FUNCTION_BLOCK FB_DiameterMovement EXTENDS FB_ObjectBase_V2
VAR_INPUT
//    Execute    :BOOL;   // True : This prog will start.
//    Abort      :BOOL;   // True : This prog will be abort.
//    Reset      :BOOL;   // True : This prog will be reset.
//    ObjectName :STRING; // Set this fb name(About it's action)
	
	bContinue:BOOL;
	
//	DiameterHorizontalCylinder 	:REFERENCE TO FB_Cylinder;	//測徑橫移氣壓缸
//	DiameterUpDownCylinder		:REFERENCE TO FB_Cylinder;	//測徑上下氣壓缸
//	DiameterClampCylinder		:REFERENCE TO FB_Cylinder; //測徑夾爪氣壓缸

	Cylinder : REFERENCE TO UNI_CylinderList;
	
END_VAR

VAR_OUTPUT
//    Busy    :BOOL;        // True : This prog is running.
//    Done    :BOOL;        // True : Command has been executed.
//    Aborted :BOOL;        // True : This prog is aborted.
//    Error   :BOOL;        // True : This prog has an error.
//    ErrorID :UINT;       // Output ErrorID
//    Status  :T_MaxString; // Output this prog status by string(255bytes)
	PickDone	:BOOL;
END_VAR

VAR
//    eState :E_MethodStatus_Basic;
//	uiExecutingStep : UDINT; // This var is used to been controll STATE_EXECUTING process.
//	uiResettingStep : UDINT;
//	uiAbortingStep : UDINT;
//	_Executed :BOOL; // Executing process completed.
//	_Error : BOOL; // FB has an error.
//	_ResetCompleted : BOOL; // FB resetting completed.
//	_AbortCompleted : BOOL; // FB aborting completed.
//	_Abort		: BOOL;
	strStatus	: STRING;
	uiResumeStep : UINT;
	tonDiameterTimeoutTwo :TON;
	
END_VAR

A00_BasicUnits();
SUPER^.A10_StateControl();

ACTION A00_BasicUnits:
tonDiameterTimeoutTwo(PT:=T#2S);
END_ACTION

METHOD GetModelState
VAR_OUTPUT
    xDone    :BOOL;
    xBusy    :BOOL;
    xError   :BOOL;
    xAborted :BOOL;
    iErrorID :UDINT;
	UniqueErrorCode : STRING;
END_VAR
xDone    := Done;
xBusy    := Busy;
xError   := Error;
xAborted := Abort;
iErrorID := ErrorID;
END_METHOD

METHOD GetName : STRING
GetName := ObjectName;
END_METHOD

METHOD  M_STATE_ABORTED
VAR_INPUT
END_VAR
ERROR :=TRUE;
Status := strStatus;

IF NOT Execute THEN
	eSTATE:=STATE_RESETTING;
END_IF

IF Execute AND Reset THEN
	uiExecutingStep :=uiResumeStep;
	eSTATE:=STATE_EXECUTING;
END_IF
END_METHOD

METHOD  M_STATE_ABORTING
VAR_INPUT
END_VAR
CASE uiAbortingStep OF
	
	
	9999:	_AbortCompleted:=TRUE;
END_CASE

IF _AbortCompleted THEN	
	eSTATE :=STATE_ABORTED;
END_IF
END_METHOD

METHOD  M_STATE_DONE
VAR_INPUT
END_VAR
Busy := FALSE;
Done:=TRUE;

IF NOT Execute THEN
	eSTATE:=STATE_RESETTING;
END_IF
END_METHOD

METHOD  M_STATE_DORMANT
VAR_INPUT
END_VAR
_Executed:=FALSE;
_Error	:=FALSE;
_Abort :=FALSE;
strStatus :='No Error';
uiResettingStep:=0;
uiExecutingStep :=0;
tonDiameterTimeoutTwo.IN:=FALSE;
Error := Busy := Done := FALSE;

IF Execute THEN
	eSTATE:=STATE_EXECUTING;
END_IF
END_METHOD

METHOD  M_STATE_ERROR
VAR_INPUT
END_VAR
ERROR :=TRUE;
Busy :=FALSE;
Done := FALSE;
Status := strStatus;
IF NOT Execute THEN	
eSTATE:=STATE_RESETTING;
END_IF
END_METHOD

METHOD  M_STATE_EXECUTING
VAR_INPUT
END_VAR
Busy :=TRUE;

CASE uiExecutingStep OF
	

0: //Standby todo : check 
	
		uiExecutingStep:=10;
10:
		
		IF Cylinder.List.fbUpCV_DiameterHoriz.xError THEN
			Cylinder.List.fbUpCV_DiameterHoriz.M_Reset();
		END_IF
		IF Cylinder.List.fbUpCV_DiameterVert.xError THEN
			Cylinder.List.fbUpCV_DiameterVert.M_Reset();
		END_IF
		IF Cylinder.List.fbUpCV_DiameterClamp.xError THEN
			Cylinder.List.fbUpCV_DiameterClamp.M_Reset();
		END_IF
		uiExecutingStep:=20;
		
20:
	Cylinder.List.fbUpCV_DiameterVert.M_Retract();
	IF Cylinder.List.fbUpCV_DiameterClamp.InFrontPosition THEN
		uiExecutingStep:=30;
	ELSE
		uiExecutingStep:=60;	
	END_IF
30:
	
	IF Cylinder.List.fbUpCV_DiameterVert.InRearPosition THEN
		Cylinder.List.fbUpCV_DiameterHoriz.M_Extend();
		uiExecutingStep:=40;
	END_IF
40:		
	IF Cylinder.List.fbUpCV_DiameterHoriz.InFrontPosition THEN
		Cylinder.List.fbUpCV_DiameterClamp.M_Retract();
		uiExecutingStep:=50;
	END_IF
50:	
	IF Cylinder.List.fbUpCV_DiameterClamp.InRearPosition THEN
		uiExecutingStep:=60;
	END_IF
	
60 : 
	Cylinder.List.fbUpCV_DiameterHoriz.M_Retract();
		uiExecutingStep:=70;
70:
	IF Cylinder.List.fbUpCV_DiameterHoriz.InRearPosition THEN
		uiExecutingStep:=1000;	
	END_IF
			
	

1000:// Pick to diameter camera position start: Clamp down
	Cylinder.List.fbUpCV_DiameterVert.M_Extend();
	uiExecutingStep:=1100;
	
1100:// wait clamp down
	tonDiameterTimeoutTwo.IN:=TRUE;
	IF 	Cylinder.List.fbUpCV_DiameterVert.InFrontPosition THEN
		tonDiameterTimeoutTwo.IN:=FALSE;
		uiExecutingStep:=1200;
	END_IF
	IF tonDiameterTimeoutTwo.Q THEN
		_Error :=TRUE;
		strStatus:='Cylinder.List.fbUpCV_DiameterVert MoveForward Timeout';
	END_IF
	
1200: // Clamp close
	Cylinder.List.fbUpCV_DiameterClamp.M_Extend();
	uiExecutingStep:=1300;

1300://wait clamp close
	tonDiameterTimeoutTwo.IN:=TRUE;
	IF 	Cylinder.List.fbUpCV_DiameterClamp.InFrontPosition THEN
		tonDiameterTimeoutTwo.IN :=FALSE;
		uiExecutingStep:=1400;
	END_IF
	IF tonDiameterTimeoutTwo.Q THEN
		_Error :=TRUE;
		strStatus:='Cylinder.List.fbUpCV_DiameterClamp M_Extend Timeout';
	END_IF
1400 : //Clamp up
	Cylinder.List.fbUpCV_DiameterVert.M_Retract();
	uiExecutingStep:=1500;	

1500:// wait clamp up
		tonDiameterTimeoutTwo.IN :=TRUE;
	IF 	Cylinder.List.fbUpCV_DiameterVert.InRearPosition THEN
		tonDiameterTimeoutTwo.IN :=FALSE;
		uiExecutingStep:=1600;
	END_IF
	IF tonDiameterTimeoutTwo.Q THEN
		_Error :=TRUE;
		strStatus:='Cylinder.List.fbUpCV_DiameterVert M_Retract Timeout';
	END_IF
1600: //Move horizontal
	Cylinder.List.fbUpCV_DiameterHoriz.M_Extend();
	uiExecutingStep:=1700;

1700://wait move horizontal
		tonDiameterTimeoutTwo.IN:=TRUE;
	IF 	Cylinder.List.fbUpCV_DiameterHoriz.InFrontPosition THEN
		tonDiameterTimeoutTwo.IN :=FALSE;
		uiExecutingStep:=1800;
	END_IF
		IF tonDiameterTimeoutTwo.Q THEN
		_Error :=TRUE;
		strStatus:='Cylinder.List.fbUpCV_DiameterHoriz M_Extend Timeout';
	END_IF

1800://Move down to diameter camera position
	Cylinder.List.fbUpCV_DiameterVert.M_Extend();
	uiExecutingStep:=1900;
	
1900:
		tonDiameterTimeoutTwo.IN:=TRUE;
	IF 	Cylinder.List.fbUpCV_DiameterVert.InFrontPosition THEN
		tonDiameterTimeoutTwo.IN :=FALSE;
		uiExecutingStep:=2000;
	END_IF	
	IF tonDiameterTimeoutTwo.Q THEN
		_Error :=TRUE;
		strStatus:='Cylinder.List.fbUpCV_DiameterVert M_Extend Timeout';
	END_IF

2000: 
	PickDone :=TRUE;
	IF bContinue THEN
		PickDone :=FALSE;
		uiExecutingStep:=5000;
	END_IF

5000: // Place needle back to box start
	Cylinder.List.fbUpCV_DiameterVert.M_Retract();
	uiExecutingStep:=5100;
	
5100:// wait clamp down
	tonDiameterTimeoutTwo.IN :=TRUE;
	IF 	Cylinder.List.fbUpCV_DiameterVert.InRearPosition THEN
		tonDiameterTimeoutTwo.IN :=FALSE;
		uiExecutingStep:=5200;
	END_IF
	IF tonDiameterTimeoutTwo.Q THEN
		_Error :=TRUE;
		strStatus:='Cylinder.List.fbUpCV_DiameterVert M_Retract Timeout';
	END_IF
	
5200: 
		Cylinder.List.fbUpCV_DiameterHoriz.M_Retract();
		uiExecutingStep := 5300;

5300:
		tonDiameterTimeoutTwo.IN :=TRUE;
		IF Cylinder.List.fbUpCV_DiameterHoriz.InRearPosition THEN
			tonDiameterTimeoutTwo.IN :=FALSE;
			uiExecutingStep := 5400;
		END_IF
		IF tonDiameterTimeoutTwo.Q THEN
		_Error :=TRUE;
		strStatus:='Cylinder.List.fbUpCV_DiameterHoriz M_Retract Timeout';
		END_IF
5400 : 
		Cylinder.List.fbUpCV_DiameterVert.M_Extend();
		uiExecutingStep:=5500;

5500:
		tonDiameterTimeoutTwo.IN :=TRUE;
		IF 	Cylinder.List.fbUpCV_DiameterVert.InFrontPosition THEN
			tonDiameterTimeoutTwo.IN:=FALSE;
			uiExecutingStep:=5600;
		END_IF
		IF tonDiameterTimeoutTwo.Q THEN
		_Error :=TRUE;
		strStatus:='Cylinder.List.fbUpCV_DiameterVert M_Extend Timeout';
		END_IF
5600: 
		Cylinder.List.fbUpCV_DiameterClamp.M_Retract();
		uiExecutingStep := 5700;
5700:	
		tonDiameterTimeoutTwo.IN :=TRUE;
		IF Cylinder.List.fbUpCV_DiameterClamp.InRearPosition THEN
			tonDiameterTimeoutTwo.IN :=FALSE;
			uiExecutingStep :=5800;
		END_IF
		IF tonDiameterTimeoutTwo.Q THEN
		_Error :=TRUE;
		strStatus:='Cylinder.List.fbUpCV_DiameterClamp M_Retract Timeout';
		END_IF
5800:
		Cylinder.List.fbUpCV_DiameterVert.M_Retract();
		 uiExecutingStep := 5900;
5900:
		tonDiameterTimeoutTwo.IN :=TRUE;
		IF Cylinder.List.fbUpCV_DiameterVert.InRearPosition THEN
			tonDiameterTimeoutTwo.IN :=FALSE;
		uiExecutingStep :=6000;
		END_IF
		IF tonDiameterTimeoutTwo.Q THEN
		_Error :=TRUE;
		strStatus:='Cylinder.List.fbUpCV_DiameterVert M_Retract Timeout';
		END_IF
6000:
		_Executed:= TRUE;





END_CASE
	
IF NOT Execute THEN
	eState:=STATE_RESETTING;
END_IF
IF _Error THEN
	eState:=STATE_ERROR;
END_IF
IF _Abort THEN
	eSTATE:=STATE_ABORTING;
END_IF
IF _Executed THEN
	eSTATE:=STATE_Done;
END_IF
END_METHOD

METHOD  M_STATE_RESETTING
VAR_INPUT
END_VAR
Error :=FALSE;
Done :=FALSE;
Busy := FALSE;


CASE uiResettingStep OF
	0 : 
		
		IF Cylinder.List.fbUpCV_DiameterHoriz.xError THEN
			Cylinder.List.fbUpCV_DiameterHoriz.M_Reset();
		END_IF
		IF Cylinder.List.fbUpCV_DiameterVert.xError THEN
			Cylinder.List.fbUpCV_DiameterVert.M_Reset();
		END_IF
		IF Cylinder.List.fbUpCV_DiameterClamp.xError THEN
			Cylinder.List.fbUpCV_DiameterClamp.M_Reset();
		END_IF
		uiResettingStep:=100;
		
	100:
		Cylinder.List.fbUpCV_DiameterVert.M_Retract();
		IF Cylinder.List.fbUpCV_DiameterClamp.InFrontPosition THEN
			uiResettingStep:=1000;
		ELSE
			uiResettingStep:=2000;	
		END_IF
	1000:
			
			IF Cylinder.List.fbUpCV_DiameterVert.InRearPosition THEN
				Cylinder.List.fbUpCV_DiameterHoriz.M_Extend();
				uiResettingStep:=1200;
			END_IF
	1200:		
			IF Cylinder.List.fbUpCV_DiameterHoriz.InFrontPosition THEN
				Cylinder.List.fbUpCV_DiameterClamp.M_Retract();
				uiResettingStep:=1300;
			END_IF
	1300:	
			IF Cylinder.List.fbUpCV_DiameterClamp.InRearPosition THEN
				uiResettingStep:=2000;
			END_IF
		
	2000 : 
			Cylinder.List.fbUpCV_DiameterHoriz.M_Retract();
				uiResettingStep:=2100;
	2100:
			IF Cylinder.List.fbUpCV_DiameterHoriz.InRearPosition THEN
				uiResettingStep:=9999;	
			END_IF
			
	9999:
		_ResetCompleted:=TRUE;
END_CASE
IF _ResetCompleted THEN
	eSTATE:=STATE_DORMANT;
END_IF
END_METHOD

END_FUNCTION_BLOCK

(* stored: Version 1.1.0.1, ProductVersion 3.1.4024.13
   POU FB_DiameterMovement: Id {5e49581e-19d4-47b9-9f67-813b2bed0ad5}, SpecialFunc None
   Folder STATE: Id {7724f639-9e7d-4988-980b-67021191a50f}
   Action A00_BasicUnits: Id {a35f34a2-2c35-4595-85bd-dd08cd46da09}
   Method GetModelState: Id {b059352f-f16e-4465-886b-930f2788111d}
   Method GetName: Id {4fc5ebf8-b8f1-4784-9a03-4ed9b9696696}
   Method M_STATE_ABORTED: Id {1eb66387-3b64-4807-892e-9f38231d5df1}
   Method M_STATE_ABORTING: Id {76cfc40e-8b02-43b9-b05d-e25adf39aa3b}
   Method M_STATE_DONE: Id {a5b57322-7bff-4937-8390-e8fd1c911d84}
   Method M_STATE_DORMANT: Id {5bf6fd3f-53ef-469a-b951-ae1c0640be83}
   Method M_STATE_ERROR: Id {6ede5fb2-605d-4718-a181-faa861654d7f}
   Method M_STATE_EXECUTING: Id {5864997d-dc49-4b0d-a74d-c3a3fca87085}
   Method M_STATE_RESETTING: Id {288044f8-b29d-4e42-b069-ce07fc47667e} *)
